Staubli VAL3: onF3Event.pgx

program onF3Event(bool& x_bSave[])
  local string l_sMessage
  local num l_nActualProg
  local string l_sButton[2]
  local bool l_bYes
  local bool l_bCancel
  local string l_sEmpty
  local num i
begin
  // look if the bButton is enable
  if bButton[2]
    if x_bSave
      call language:message(l_sMessage,-1)
      // get the yes_no button Key
      call language:getYesNo(l_sButton)
      // ask the question
      call use:yes_no_cancel(l_sMessage,l_sButton,l_bYes,l_bCancel)
      if l_bYes
        call saveIt(x_bSave)
      endIf
    endIf
    // check if the cancel button has been pressed
    if !l_bCancel
      l_sEmpty=""
      call loadPage("Disk://instruction/inputOutput/page_inOut",l_sEmpty)
      call prog:load(sProgram,i)
      if i!=0
        // show the error message
        call language:message(l_sMessage,-7)
        popUpMsg(l_sMessage+" PROG "+sProgram+", "+toString("",i))
      endIf
      // return to the page
      logMsg("[KERNEL] INTERFACE:Page Edit Program: "+sProgram)
      call buildList()
    endIf
  endIf
end
